{attribute 'linkalways'} 
{attribute 'no_explicit_call' := 'This FB is a CLASS and must be accessed using methods or properties'}
{attribute 'enable_dynamic_creation'}
FUNCTION_BLOCK Node_F_VN_DrawRectangle_TcVnRectangle_UDINT EXTENDS VisionNode
VAR
    stRectangle : _TcVnRectangle_UDINT;
    ipDestImage : _ITcVnImage;
    aColor : _TcVnVector4_LREAL;
    nThickness : _DINT(1);
    hrPrev : _HRESULT(S_OK);
	hresult : _HRESULT(S_OK);
END_VAR

METHOD PUBLIC  Clone : I_Node
VAR
	pNode : POINTER TO Node_F_VN_DrawRectangle_TcVnRectangle_UDINT;
END_VAR
pNode := __NEW(Node_F_VN_DrawRectangle_TcVnRectangle_UDINT);
Clone := pNode^;
END_METHOD

METHOD FB_init : BOOL
VAR_INPUT
	bInitRetains : BOOL; // if TRUE, the retain variables are initialized (warm start / cold start)
	bInCopyCode : BOOL;  // if TRUE, the instance afterwards gets moved into the copy code (online change)
END_VAR
AddInput('stRectangle', stRectangle);
AddInput('ipDestImage', ipDestImage);
AddInput('aColor', aColor);
AddParameter('nThickness', nThickness);
AddInput('hrPrev', hrPrev);
AddOutput('ipDestImage', ipDestImage);
AddOutput('hresult',hresult);
END_METHOD

METHOD PROTECTED OnExecute
hresult.Value := F_VN_DrawRectangle_TcVnRectangle_UDINT(
    stRectangle := stRectangle.Value,
	ipDestImage := ipDestImage.Value,
    aColor := aColor.Value,
    nThickness := nThickness.Value,
	hrPrev:= hrPrev.Value);
END_METHOD

METHOD PUBLIC PreExecutionCheck
VAR_INPUT
	Check : I_PreExecutionChecks;
END_VAR
Check.IsTrue(ipDestImage.IsValid, 'ipDestImage must contain an image');
Check.IsTrue(nThickness.Value <> 0, 'nThickness must be non-zero');
END_METHOD

END_FUNCTION_BLOCK

(* stored: Version 1.1.0.1, ProductVersion 3.1.4024.15
   POU Node_F_VN_DrawRectangle_TcVnRectangle_UDINT: Id {d53ca39a-dbec-03bd-0cfc-1a275264cdae}, SpecialFunc None
   Folder Constructor: Id {71ba0c90-1619-09ad-2bb9-b0210c0b2481}
   Method Clone: Id {833bf71b-40f2-0a0a-10f3-b56fa0d9df6f}
   Method FB_init: Id {f5db2bb8-84cf-0f96-1080-3ae253bffe50}
   Method OnExecute: Id {48cd1a10-a2db-063f-1f15-04443daaf726}
   Method PreExecutionCheck: Id {b064442f-dc07-0c9e-1189-a2aa5a13054c} *)
